INTERFACE I_LightControl

METHOD M_Reset : BOOL
VAR_INPUT
END_VAR
END_METHOD

METHOD M_Set : BOOL
VAR_INPUT
END_VAR
END_METHOD

PROPERTY nAddress : dint
GET
END_GET
SET
END_SET
END_PROPERTY

PROPERTY nIlluminance : real
GET
END_GET
SET
END_SET
END_PROPERTY

END_INTERFACE

(* stored: Version 1.1.0.1, ProductVersion 3.1.4022.18
   Itf I_LightControl: Id {a69c5011-7319-4bf8-a869-2c7adb65cb07}
   Method M_Reset: Id {b47b4758-e09c-48dd-9b75-d61a69cc8597}
   Method M_Set: Id {71c054e3-b394-4398-8263-4ad96451bf8a}
   Property nAddress: Id {27008ca9-1135-4ca4-8b67-90dc83916b6e}
   Get Get: Id {9bbbc337-3207-46af-bf8d-e5ba54c0ffbf}
   Set Set: Id {c8ecdddf-f965-4041-a142-1e8bbb24851a}
   Property nIlluminance: Id {43322e26-a80a-4655-9558-c79d31ec8fe3}
   Get Get: Id {a97ce1bc-6f29-4456-bde2-11640ccee9bf}
   Set Set: Id {8959a0fc-3933-4f9d-9755-4bf43517701b} *)
